// TIA Portal V20 export
DATA_BLOCK "OperatorPrompts"   // DB123
// stored: Access Published, MemoryReserve 100
   VAR
      triggers { ExternalAccessible := 'False'; ExternalVisible := 'False'; ExternalWritable := 'False'} : Array[1..63] of Bool;
      activeOperatorPrompt { ExternalWritable := 'False'} : Int;
      ack : Bool;
   END_VAR
BEGIN
END_DATA_BLOCK
